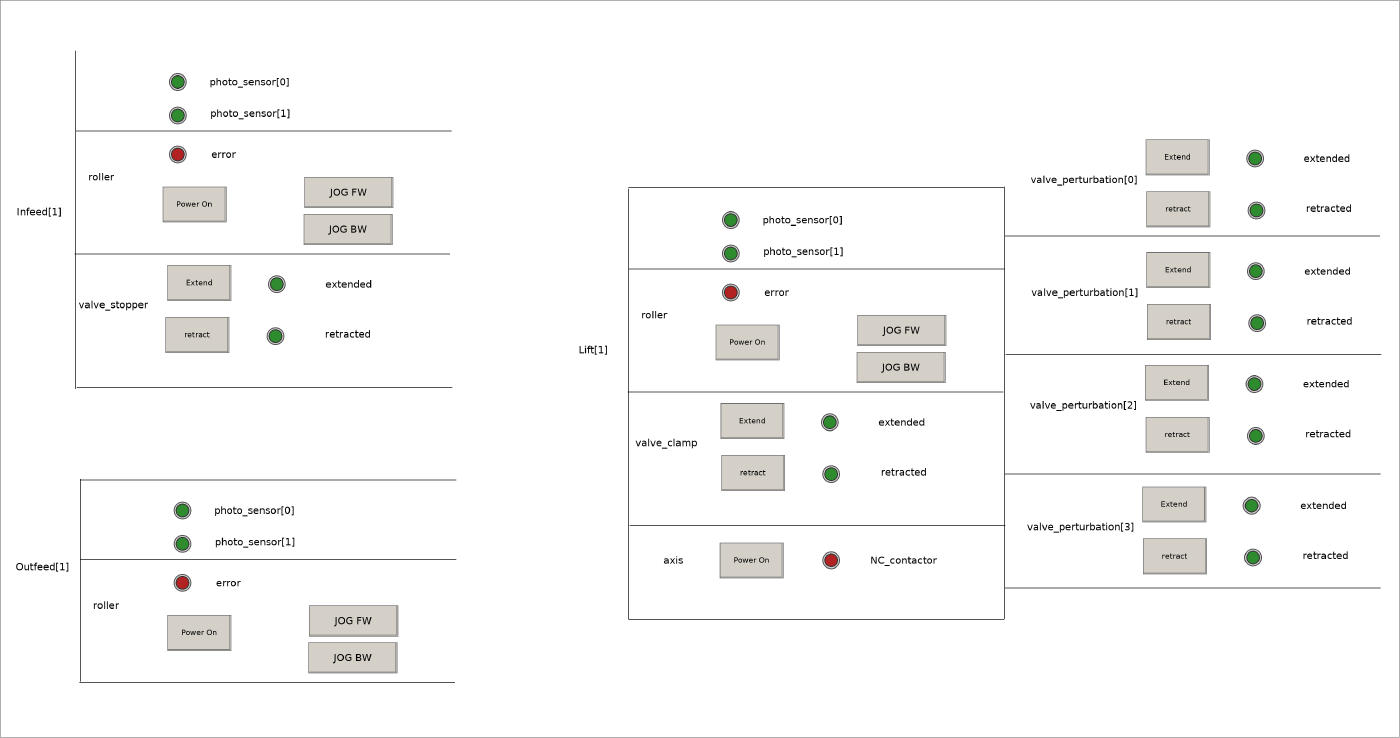
VISUALIZATION v_rem_1  // 2048x1080
VAR_IN_OUT
	dIO_ReM		: Replenishment_Module;
END_VAR
    Lamp1 (245,105 30x30), variable: dIO_ReM.infeed[1].photo_sensor[0].debounced_input.Q, style: Lamp-Lamp1-Green
    Lamp1 (245,154 30x30), variable: dIO_ReM.infeed[1].photo_sensor[1].debounced_input.Q, style: Lamp-Lamp1-Green
    Label (299,107 132x26), "photo_sensor[0]"
    Label (300,153 132x26), "photo_sensor[1]"
    Label (19,297 77x26), "Infeed[1]"
    Lamp1 (245,211 30x30), variable: dIO_ReM.infeed[1].roller.err, style: Lamp-Lamp1-Red
    Label (261,213 132x26), "error"
    Label (82,246 132x26), "roller"
    Line (111,191) (660,191)
    Line (110,74) (110,569)
    Label (100,433 132x26), "valve_stopper"
    Button (445,259 130x45), "JOG FW", colour toggle: dIO_ReM.infeed[1].roller.forward
        OnMouseDown: execute { dIO_ReM.infeed[1].roller.forward := TRUE; }
        OnMouseUp: execute { dIO_ReM.infeed[1].roller.forward := FALSE; }
    Button (444,313 130x45), "JOG BW", colour toggle: dIO_ReM.infeed[1].roller.backward
        OnMouseDown: execute { dIO_ReM.infeed[1].roller.backward := TRUE; }
        OnMouseUp: execute { dIO_ReM.infeed[1].roller.backward := FALSE; }
    Button (238,273 93x52), "Power On", colour toggle: dIO_ReM.infeed[1].roller.Power
        toggle dIO_ReM.infeed[1].roller.Power
    Button (245,388 93x52), "Extend", colour toggle: dIO_ReM.infeed[1].valve_stopper.extend
        OnMouseDown: execute { dIO_ReM.infeed[1].valve_stopper.extend := TRUE; dIO_ReM.infeed[1].valve_stopper.retract := FALSE; }
    Button (242,464 93x52), "retract", colour toggle: dIO_ReM.infeed[1].valve_stopper.retract
        OnMouseDown: execute { dIO_ReM.infeed[1].valve_stopper.extend := FALSE; dIO_ReM.infeed[1].valve_stopper.retract := TRUE; }
    Lamp1 (390,401 30x30), variable: dIO_ReM.infeed[1].valve_stopper.extended, style: Lamp-Lamp1-Green
    Lamp1 (388,477 30x30), variable: dIO_ReM.infeed[1].valve_stopper.retracted, style: Lamp-Lamp1-Green
    Label (444,403 132x26), "extended"
    Label (443,476 132x26), "retracted"
    Line (109,371) (658,371)
    Line (112,567) (661,567)
    Lamp1 (252,732 30x30), variable: dIO_ReM.outfeed[1].photo_sensor[0].debounced_input.Q, style: Lamp-Lamp1-Green
    Lamp1 (252,781 30x30), variable: dIO_ReM.outfeed[1].photo_sensor[1].debounced_input.Q, style: Lamp-Lamp1-Green
    Label (306,734 132x26), "photo_sensor[0]"
    Label (307,780 132x26), "photo_sensor[1]"
    Label (22,816 80x27), "Outfeed[1]"
    Lamp1 (252,838 30x30), variable: dIO_ReM.outfeed[1].roller.err, style: Lamp-Lamp1-Red
    Label (268,840 132x26), "error"
    Label (89,873 132x26), "roller"
    Line (118,818) (667,818)
    Line (117,701) (117,997)
    Button (452,886 130x45), "JOG FW", colour toggle: dIO_ReM.outfeed[1].roller.forward
        OnMouseDown: execute { dIO_ReM.outfeed[1].roller.forward := TRUE; }
        OnMouseUp: execute { dIO_ReM.outfeed[1].roller.forward := FALSE; }
    Button (451,940 130x45), "JOG BW", colour toggle: dIO_ReM.outfeed[1].roller.backward
        OnMouseDown: execute { dIO_ReM.outfeed[1].roller.backward := TRUE; }
        OnMouseUp: execute { dIO_ReM.outfeed[1].roller.backward := FALSE; }
    Button (245,900 93x52), "Power On", colour toggle: dIO_ReM.outfeed[1].roller.Power
        toggle dIO_ReM.outfeed[1].roller.Power
    Line (116,998) (665,998)
    Line (118,702) (667,702)
    Lamp1 (1054,307 30x30), variable: dIO_ReM.lift[1].photo_sensor[0].debounced_input.Q, style: Lamp-Lamp1-Green
    Lamp1 (1054,356 30x30), variable: dIO_ReM.lift[1].photo_sensor[1].debounced_input.Q, style: Lamp-Lamp1-Green
    Label (1108,309 132x26), "photo_sensor[0]"
    Label (1109,355 132x26), "photo_sensor[1]"
    Label (828,499 80x26), "Lift[1]"
    Lamp1 (1054,413 30x30), variable: dIO_ReM.lift[1].roller.err, style: Lamp-Lamp1-Red
    Label (1070,415 132x26), "error"
    Label (891,448 132x26), "roller"
    Line (920,393) (1469,393)
    Line (919,276) (919,906)
    Label (909,635 132x26), "valve_clamp"
    Button (1254,461 130x45), "JOG FW", colour toggle: dIO_ReM.lift[1].roller.forward
        OnMouseDown: execute { dIO_ReM.lift[1].roller.forward := TRUE; }
        OnMouseUp: execute { dIO_ReM.lift[1].roller.forward := FALSE; }
    Button (1253,515 130x45), "JOG BW", colour toggle: dIO_ReM.lift[1].roller.backward
        OnMouseDown: execute { dIO_ReM.lift[1].roller.backward := TRUE; }
        OnMouseUp: execute { dIO_ReM.lift[1].roller.backward := FALSE; }
    Button (1047,475 93x52), "Power On", colour toggle: dIO_ReM.lift[1].roller.Power
        toggle dIO_ReM.lift[1].roller.Power
    Button (1054,590 93x52), "Extend", colour toggle: dIO_ReM.lift[1].valve_clamp.extend
        OnMouseDown: execute { dIO_ReM.lift[1].valve_clamp.extend := TRUE; dIO_ReM.lift[1].valve_clamp.retract := FALSE; }
    Button (1055,666 93x52), "retract", colour toggle: dIO_ReM.lift[1].valve_clamp.retract
        OnMouseDown: execute { dIO_ReM.lift[1].valve_clamp.extend := FALSE; dIO_ReM.lift[1].valve_clamp.retract := TRUE; }
    Lamp1 (1199,603 30x30), variable: dIO_ReM.lift[1].valve_clamp.extended, style: Lamp-Lamp1-Green
    Lamp1 (1201,679 30x30), variable: dIO_ReM.lift[1].valve_clamp.retracted, style: Lamp-Lamp1-Green
    Label (1253,605 132x26), "extended"
    Label (1256,678 132x26), "retracted"
    Line (918,573) (1467,573)
    Line (921,769) (1470,769)
    Label (1506,250 160x26), "valve_perturbation[0]"
    Button (1676,204 93x52), "Extend", colour toggle: dIO_ReM.lift[1].valve_perturbation[0].extend
        OnMouseDown: execute { dIO_ReM.lift[1].valve_perturbation[0].extend := TRUE; dIO_ReM.lift[1].valve_perturbation[0].retract := FALSE; }
    Button (1677,280 93x52), "retract", colour toggle: dIO_ReM.lift[1].valve_perturbation[0].retract
        OnMouseDown: execute { dIO_ReM.lift[1].valve_perturbation[0].extend := FALSE; dIO_ReM.lift[1].valve_perturbation[0].retract := TRUE; }
    Lamp1 (1821,217 30x30), variable: dIO_ReM.lift[1].valve_perturbation[0].extended, style: Lamp-Lamp1-Green
    Lamp1 (1823,293 30x30), variable: dIO_ReM.lift[1].valve_perturbation[0].retracted, style: Lamp-Lamp1-Green
    Label (1875,219 132x26), "extended"
    Label (1878,292 132x26), "retracted"
    Label (1507,415 160x26), "valve_perturbation[1]"
    Button (1677,369 93x52), "Extend", colour toggle: dIO_ReM.lift[1].valve_perturbation[1].extend
        OnMouseDown: execute { dIO_ReM.lift[1].valve_perturbation[1].extend := TRUE; dIO_ReM.lift[1].valve_perturbation[1].retract := FALSE; }
    Button (1678,445 93x52), "retract", colour toggle: dIO_ReM.lift[1].valve_perturbation[1].retract
        OnMouseDown: execute { dIO_ReM.lift[1].valve_perturbation[1].extend := FALSE; dIO_ReM.lift[1].valve_perturbation[1].retract := TRUE; }
    Lamp1 (1822,382 30x30), variable: dIO_ReM.lift[1].valve_perturbation[1].extended, style: Lamp-Lamp1-Green
    Lamp1 (1824,458 30x30), variable: dIO_ReM.lift[1].valve_perturbation[1].retracted, style: Lamp-Lamp1-Green
    Label (1876,384 132x26), "extended"
    Label (1879,457 132x26), "retracted"
    Label (1505,580 160x26), "valve_perturbation[2]"
    Button (1675,534 93x52), "Extend", colour toggle: dIO_ReM.lift[1].valve_perturbation[2].extend
        OnMouseDown: execute { dIO_ReM.lift[1].valve_perturbation[2].extend := TRUE; dIO_ReM.lift[1].valve_perturbation[2].retract := FALSE; }
    Button (1676,610 93x52), "retract", colour toggle: dIO_ReM.lift[1].valve_perturbation[2].retract
        OnMouseDown: execute { dIO_ReM.lift[1].valve_perturbation[2].extend := FALSE; dIO_ReM.lift[1].valve_perturbation[2].retract := TRUE; }
    Lamp1 (1820,547 30x30), variable: dIO_ReM.lift[1].valve_perturbation[2].extended, style: Lamp-Lamp1-Green
    Lamp1 (1822,623 30x30), variable: dIO_ReM.lift[1].valve_perturbation[2].retracted, style: Lamp-Lamp1-Green
    Label (1874,549 132x26), "extended"
    Label (1877,622 132x26), "retracted"
    Label (1501,758 160x26), "valve_perturbation[3]"
    Button (1671,712 93x52), "Extend", colour toggle: dIO_ReM.lift[1].valve_perturbation[3].extend
        OnMouseDown: execute { dIO_ReM.lift[1].valve_perturbation[3].extend := TRUE; dIO_ReM.lift[1].valve_perturbation[3].retract := FALSE; }
    Button (1672,788 93x52), "retract", colour toggle: dIO_ReM.lift[1].valve_perturbation[3].retract
        OnMouseDown: execute { dIO_ReM.lift[1].valve_perturbation[3].extend := FALSE; dIO_ReM.lift[1].valve_perturbation[3].retract := TRUE; }
    Lamp1 (1816,725 30x30), variable: dIO_ReM.lift[1].valve_perturbation[3].extended, style: Lamp-Lamp1-Green
    Lamp1 (1818,801 30x30), variable: dIO_ReM.lift[1].valve_perturbation[3].retracted, style: Lamp-Lamp1-Green
    Label (1870,727 132x26), "extended"
    Label (1873,800 132x26), "retracted"
    Line (1469,273) (1469,906)
    Line (1469,345) (2018,345)
    Line (1471,518) (2020,518)
    Line (1470,693) (2019,693)
    Line (1470,860) (2019,860)
    Line (919,274) (1468,274)
    Line (919,906) (1468,906)
    Label (1256,807 132x26), "NC_contactor"
    Label (919,807 132x26), "axis"
    Button (1053,794 93x52), "Power On", colour toggle: dIO_ReM.lift[1].power_axis
        toggle dIO_ReM.lift[1].power_axis
    Lamp1 (1201,805 30x30), variable: dIO_ReM.lift[1].contactor_axis, style: Lamp-Lamp1-Red
END_VISUALIZATION

(* stored: Version 1.1.0.1, ProductVersion 3.1.4024.12
   Visu v_rem_1: Id {be35b70f-80af-4525-8f99-723995dfe330} *)
